INTERFACE I_RpcServer

METHOD PUBLIC RegisterApi
VAR_INPUT
	RpcApi : I_RpcApi;
END_VAR
END_METHOD

METHOD PUBLIC RegisterAsynchronousRpcHandler
VAR_INPUT
	MethodName : T_MAXSTRING;
	Handler : I_AsynchronousRpcHandler;
END_VAR
END_METHOD

METHOD PUBLIC RegisterSynchronousRpcHandler
VAR_INPUT
	MethodName : T_MAXSTRING;
	Handler : I_SynchronousRpcHandler;
END_VAR
END_METHOD

END_INTERFACE

(* stored: Version 1.1.0.1, ProductVersion 3.1.4024.12
   Itf I_RpcServer: Id {3249790d-2361-4909-9f7a-771c2ba70619}
   Method RegisterApi: Id {1683fa06-5bc8-42bf-97be-84865033b985}
   Method RegisterAsynchronousRpcHandler: Id {c7ede9aa-6e51-466a-80ea-5a4569d1c9eb}
   Method RegisterSynchronousRpcHandler: Id {e9370da5-05df-4cae-8260-53b6cf2d257e} *)
